// 1-WORD divide to 2-USINT
FUNCTION WORD_TO_USINT_Bit_1 : outWord
VAR_INPUT
	nOutput : WORD;
END_VAR
VAR
	outWord : outWord;
END_VAR

outWord.Lower := TO_USINT(nOutput); //Lower Bits
outWord.Upper := TO_USINT(SHR(nOutput, 8)); //Uppper Bits
WORD_TO_USINT_Bit := outWord;

END_FUNCTION

(* stored: Version 1.1.0.1, ProductVersion 3.1.4024.12
   POU WORD_TO_USINT_Bit_1: Id {e59653a8-d9f4-410d-ae09-69d44d20bee9}, SpecialFunc None *)
